VAR_GLOBAL
    bInput    AT %I0.0 : BOOL;
    nAnalog   AT %I2   : INT;
    bOutput   AT %Q0.0 : BOOL;
    nSetpoint AT %Q4   : DINT;
END_VAR

(* stored: Version 1.1.0.1, ProductVersion 3.1.4024.16
   GVL GVL_Syntax_Address: Id {c0f546e2-e66f-4137-95fc-87f0e029462f} *)
